FUNCTION_BLOCK FB_BadFormat
VAR
END_VAR

END_FUNCTION_BLOCK

(* stored: Version 1.1.0.1, ProductVersion 3.1.4024.12
   POU FB_BadFormat: Id {12345678-1234-1234-1234-123456789abc}, SpecialFunc None *)
